(* CoDeSys 2.3 export: DEV7SJ6x0.EXP *)

(* POU SGL_Sismored/Sismored 4.0/Imported/Dev7SJ6x0, FAI *)
FUNCTION_BLOCK Dev7SJ6x0
VAR_INPUT
xFirstCycle        :   BOOL;
iSequenceOrder     :   INT;
sProtocol          :   STRING;
eState             :   eStates;
eAction            :   eActions;
wMeasure1, wMeasure2, wMeasure3, wMeasure4, wMeasure5, wMeasure6, wMeasure7, wMeasure8, wMeasure9, wMeasure10, wMeasure11: WORD;
xSaveMeasure1, xSaveMeasure2, xSaveMeasure3, xSaveMeasure4, xSaveMeasure5, xSaveMeasure6, xSaveMeasure7, xSaveMeasure8, xSaveMeasure9, xSaveMeasure10, xSaveMeasure11: BOOL;
sNameMeasure1, sNameMeasure2, sNameMeasure3, sNameMeasure4, sNameMeasure5, sNameMeasure6, sNameMeasure7, sNameMeasure8, sNameMeasure9, sNameMeasure10, sNameMeasure11: STRING;
xState1, xState2, xState3, xState4, xState5, xState6, xState7, xState8, xState9, xState10, xState11, xState12, xState13, xState14, xState15, xState16, xState17, xState18, xState19, xState20, xState21, xState22, xState23, xState24, xState25, xState26, xState27, xState28, xState29, xState30, xState31, xState32, xState33, xState34, xState35, xState36, xState37, xState38, xState39, xState40, xState41, xState42, xState43, xState44, xState45, xState46, xState47, xState48: BOOL;
xSaveState1, xSaveState2, xSaveState3, xSaveState4, xSaveState5, xSaveState6, xSaveState7, xSaveState8, xSaveState9, xSaveState10, xSaveState11, xSaveState12, xSaveState13, xSaveState14, xSaveState15, xSaveState16, xSaveState17, xSaveState18, xSaveState19, xSaveState20, xSaveState21, xSaveState22, xSaveState23, xSaveState24, xSaveState25, xSaveState26, xSaveState27, xSaveState28, xSaveState29, xSaveState30, xSaveState31, xSaveState32, xSaveState33, xSaveState34, xSaveState35, xSaveState36, xSaveState37, xSaveState38, xSaveState39, xSaveState40, xSaveState41, xSaveState42, xSaveState43, xSaveState44, xSaveState45, xSaveState46, xSaveState47, xSaveState48: BOOL;
sNameState1, sNameState2, sNameState3, sNameState4, sNameState5, sNameState6, sNameState7, sNameState8, sNameState9, sNameState10, sNameState11, sNameState12, sNameState13, sNameState14, sNameState15, sNameState16, sNameState17, sNameState18, sNameState19, sNameState20, sNameState21, sNameState22, sNameState23, sNameState24, sNameState25, sNameState26, sNameState27, sNameState28, sNameState29, sNameState30, sNameState31, sNameState32, sNameState33, sNameState34, sNameState35, sNameState36, sNameState37, sNameState38, sNameState39, sNameState40, sNameState41, sNameState42, sNameState43, sNameState44, sNameState45, sNameState46, sNameState47, sNameState48: STRING;
xCommand1, xCommand2, xCommand3, xCommand4, xCommand5, xCommand6, xCommand7, xCommand8, xCommand9: BOOL;
xSaveCommand1, xSaveCommand2, xSaveCommand3, xSaveCommand4, xSaveCommand5, xSaveCommand6, xSaveCommand7, xSaveCommand8, xSaveCommand9: BOOL;
sNameCommand1, sNameCommand2, sNameCommand3, sNameCommand4, sNameCommand5, sNameCommand6, sNameCommand7, sNameCommand8, sNameCommand9: STRING;
END_VAR
VAR_OUTPUT
wMeasureOutput1, wMeasureOutput2, wMeasureOutput3, wMeasureOutput4, wMeasureOutput5, wMeasureOutput6, wMeasureOutput7, wMeasureOutput8, wMeasureOutput9, wMeasureOutput10, wMeasureOutput11: WORD;
xStateOutput1, xStateOutput2, xStateOutput3, xStateOutput4, xStateOutput5, xStateOutput6, xStateOutput7, xStateOutput8, xStateOutput9, xStateOutput10, xStateOutput11, xStateOutput12, xStateOutput13, xStateOutput14, xStateOutput15, xStateOutput16, xStateOutput17, xStateOutput18, xStateOutput19, xStateOutput20, xStateOutput21, xStateOutput22, xStateOutput23, xStateOutput24, xStateOutput25, xStateOutput26, xStateOutput27, xStateOutput28, xStateOutput29, xStateOutput30, xStateOutput31, xStateOutput32, xStateOutput33, xStateOutput34, xStateOutput35, xStateOutput36, xStateOutput37, xStateOutput38, xStateOutput39, xStateOutput40, xStateOutput41, xStateOutput42, xStateOutput43, xStateOutput44, xStateOutput45, xStateOutput46, xStateOutput47, xStateOutput48: BOOL;
xCommandOutput1, xCommandOutput2, xCommandOutput3, xCommandOutput4, xCommandOutput5, xCommandOutput6, xCommandOutput7, xCommandOutput8, xCommandOutput9: BOOL;
END_VAR
VAR
inst0Rtu11word7SJ6xm0 : Rtu11word7SJ6xm0;
inst0Rtu48bool7SJ6xs0 : Rtu48bool7SJ6xs0;
inst0Rtu9bool7SJ6xc0 : Rtu9bool7SJ6xc0;
END_VAR
(* body not read: x-want_COMMENT *)
END_FUNCTION_BLOCK
